// TIA Portal project "Item Queuing" (V16)

(* hardware
DEVICE "S7300/ET200M station_1"  S7-300 station
   slot 0: "Rail_0"  Rail  6ES7 390-1***0-0AA0
   slot 2: "PLC_1"  CPU 312  6ES7 312-1AE13-0AB0  V2.6
      slot 0: "MPI interface_1"  X1
*)

// ===== PLC "PLC_1"  CPU 312 =====

VAR_GLOBAL   // PLC tag table "Default tag table"
   "Emergncy" AT %I0.1 : Bool;
   "Item sensor" AT %I0.2 : Bool;
   "Sensor - 1" AT %I0.3 : Bool;
   "Sensor - 2" AT %I0.4 : Bool;
   "Exit - Sensor" AT %I0.5 : Bool;
   "Conv - 0" AT %Q0.0 : Bool;
   "Conv - 1" AT %Q0.1 : Bool;
   "Conv - 2" AT %Q0.2 : Bool;
   "Sensor - 3" AT %I0.6 : Bool;
   "T1" AT %M5.5 : Bool;
   "T2" AT %M6.6 : Bool;
END_VAR

ORGANIZATION_BLOCK "Main"   // OB1, LAD
TITLE = "Main Program Sweep (Cycle)"
{ S7_Optimized_Access := 'FALSE' }
VERSION : 0.1
   VAR_TEMP
      OB1_EV_CLASS : Byte;   // Bits 0-3 = 1 (Coming event), Bits 4-7 = 1 (Event class 1)
      OB1_SCAN_1 : Byte;   // 1 (Cold restart scan 1 of OB 1), 3 (Scan 2-n of OB 1)
      OB1_PRIORITY : Byte;   // Priority of OB Execution
      OB1_OB_NUMBR : Byte;   // 1 (Organization block 1, OB1)
      OB1_RESERVED_1 : Byte;   // Reserved for system
      OB1_RESERVED_2 : Byte;   // Reserved for system
      OB1_PREV_CYCLE : Int;   // Cycle time of previous OB1 scan (milliseconds)
      OB1_MIN_CYCLE : Int;   // Minimum cycle time of OB1 (milliseconds)
      OB1_MAX_CYCLE : Int;   // Maximum cycle time of OB1 (milliseconds)
      OB1_DATE_TIME : Date_And_Time;   // Date and time OB1 started
   END_VAR
   VAR_TEMP   // added for the SCL form of the ladder/FBD networks
      _w1 : Bool;
   END_VAR
BEGIN

REGION Network 1
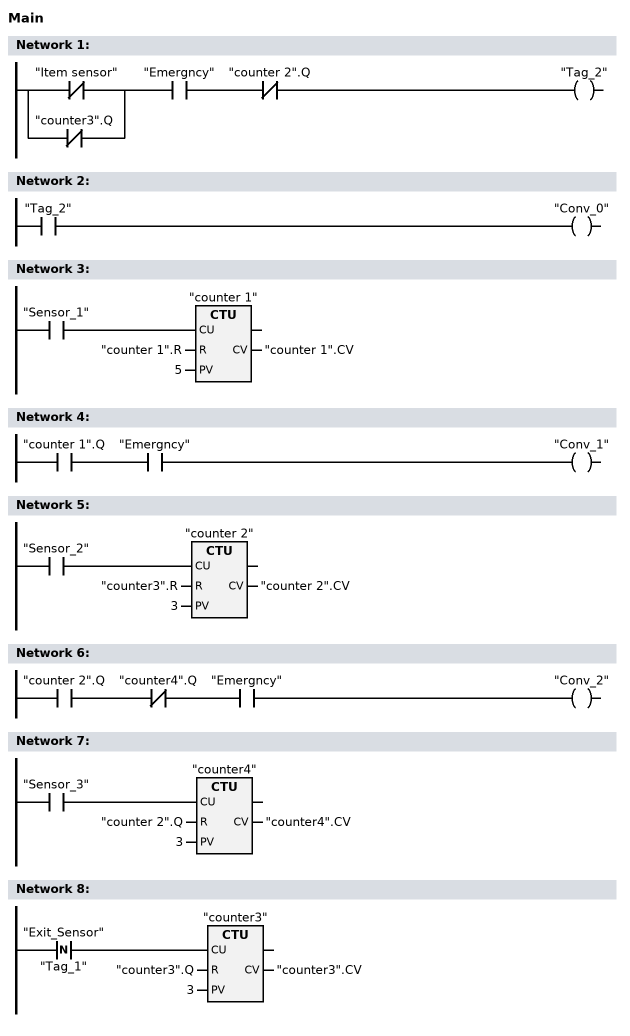
   RUNG wire#powerrail
      I_Contact( "Item sensor" )
      wire#w1
      Contact( "Emergncy" )
      I_Contact( "counter 2".Q )
      Coil( "Tag_2" )
   END_RUNG
   RUNG wire#powerrail
      I_Contact( "counter3".Q )
   END_RUNG wire#w1
   // the same network as SCL:
   "Tag_2" := (NOT "Item sensor" OR NOT "counter3".Q) AND "Emergncy" AND NOT "counter 2".Q;
END_REGION

REGION Network 2
   RUNG wire#powerrail
      Contact( "Tag_2" )
      Coil( "Conv_0" )
   END_RUNG
   // the same network as SCL:
   "Conv_0" := "Tag_2";
END_REGION

REGION Network 3
   "counter 1".CTU(CU := "Sensor_1", R := "counter 1".R, PV := 5, CV => "counter 1".CV);
END_REGION

REGION Network 4
   RUNG wire#powerrail
      Contact( "counter 1".Q )
      Contact( "Emergncy" )
      Coil( "Conv_1" )
   END_RUNG
   // the same network as SCL:
   "Conv_1" := "counter 1".Q AND "Emergncy";
END_REGION

REGION Network 5
   "counter 2".CTU(CU := "Sensor_2", R := "counter3".R, PV := 3, CV => "counter 2".CV);
END_REGION

REGION Network 6
   RUNG wire#powerrail
      Contact( "counter 2".Q )
      I_Contact( "counter4".Q )
      Contact( "Emergncy" )
      Coil( "Conv_2" )
   END_RUNG
   // the same network as SCL:
   "Conv_2" := "counter 2".Q AND NOT "counter4".Q AND "Emergncy";
END_REGION

REGION Network 7
   "counter4".CTU(CU := "Sensor_3", R := "counter 2".Q, PV := 3, CV => "counter4".CV);
END_REGION

REGION Network 8
   #_w1 := NOT "Exit_Sensor" AND "Tag_1";   // falling edge of "Exit_Sensor"
   "Tag_1" := "Exit_Sensor";
   "counter3".CTU(CU := #_w1, R := "counter3".Q, PV := 3, CV => "counter3".CV);
END_REGION
END_ORGANIZATION_BLOCK